// TIA Portal V16 export
// export: Created 2021-07-12T14:47:14.9842016Z, ExportSetting WithDefaults, DisplayName Totally Integrated Automation Portal, DisplayVersion V16, DisplayName TIA Portal Version Control Interface, DisplayVersion V16, DisplayName TIA Portal Openness, DisplayVersion V16, DisplayName STEP 7 Professional, DisplayVersion V16, DisplayName STEP 7 Safety, DisplayVersion V16, DisplayName WinCC Professional, DisplayVersion V16
DATA_BLOCK "LSimaHydTO_HydAxisDriveInterfaceTemplate"   // DB33051
TITLE = LSimaHydTO_HydAxisDriveInterfaceTemplate
{ S7_Optimized_Access := 'FALSE'; DB_Accessible_From_OPC_UA := 'FALSE' }
AUTHOR : APC_ERLF
FAMILY : LSimaHydTO
VERSION : 1.0
// stored: AutoNumber true, DBAccessibleFromOPCUA false, IsOnlyStoredInLoadMemory false, IsWriteProtectedInAS false
   VAR
      tel2 { ExternalAccessible := 'False'; ExternalVisible := 'False'; ExternalWritable := 'False'; S7_SetPoint := 'True'} : PD_TEL2;
      tel81 { ExternalAccessible := 'False'; ExternalVisible := 'False'; ExternalWritable := 'False'; S7_SetPoint := 'True'} : PD_TEL81;
   END_VAR
BEGIN
END_DATA_BLOCK
